{attribute 'qualified_only'}
{attribute 'strict'}

//-----------------------------------------------------------------------------------------
//
//                  			ENUM_Log_File_Management
//
//									Log file management 			
//-----------------------------------------------------------------------------------------
//
//Auteur: G.GOETZ (inspired by S.MANTZER)
//Création: 04.02.2026
//Dernière modification : 04.02.2026 (G.GOETZ)
//       			
//-----------------------------------------------------------------------------------------
//
//     							Liste des modifications  	
//
// 04.02.2026 (G.GOETZ) -> Création		
//-----------------------------------------------------------------------------------------

TYPE ENUM_Log_File_Management :
(
	Automatic := 1 , 
	Manual := 2 ,	
	ManualWithDelete := 3 
);
END_TYPE

(* stored: Version 1.1.0.1, ProductVersion 3.1.4024.13
   DUT ENUM_Log_File_Management: Id {38c60f07-815f-4227-8ca4-1344f343e8a2} *)
